FUNCTION FUN_AddValuleToString : STRING(490)
VAR_INPUT
	sString		:STRING(490);	// String where value is to be added
	rValue		:LREAL;			// Value to be added to string
	iNoOfDec	:INT;			// Number of decimals to be presented in the string
END_VAR
VAR
	sSeperator	:STRING(80);	// Seperator
	sValue		:STRING(80);	// String version of value
END_VAR


// Create string for value
sValue := FUN_RealToString(rValue:= rValue, iNoOfDec:= iNoOfDec);

// Replace "." character with "," character (special Elvstrøm request)
sValue := FUN_ReplaceDotWithComma(sStringIn:= sValue);

// Add seperator to string
sSeperator := ';';
CONCAT2(pSrcString1:= ADR(sString), pSrcString2:= ADR(sSeperator), pDstString:= ADR(sString), nDstSize:= 490);

// Add value to string
CONCAT2(pSrcString1:= ADR(sString), pSrcString2:= ADR(sValue), pDstString:= ADR(sString), nDstSize:= 490);

// Return string
FUN_AddValuleToString := sString;

END_FUNCTION

(* stored: Version 1.1.0.1, ProductVersion 3.1.4024.12
   POU FUN_AddValuleToString: Id {977a6f7c-d993-4d95-9b61-b9120a1bc4b3}, SpecialFunc None *)
